(* IEC 61131-3 sources: eCockpitGit/test_project/src/%F%00 Library/%F%Common Functions/%F%Time, 12 files *)

(* ---- %DUT%ATimeShow.st ---- *)
TYPE ATimeShow : STRING(19); END_TYPE

(* ---- %POU%FU_sCountUpDateTime.st ---- *)
//This function, converts passed seconds to minutes, hours, days, weeks, years, and only outputs the two biggest active time formats
//example 249 = Minutes: 4 Seconds: 9, 529385 = Days: 6 Hours: 3
// |**Version**|**Author**| **Date** |**Changes**
// | 1         | NSN      | 09-01-18 | Updated to new format
// | 1         | NSN      | 13-06-18 | Updated names and types
FUNCTION FU_sCountUpDateTime : STRING(24)
VAR_INPUT
	dwSeconds	:DWORD;		//Input seconds
END_VAR
VAR
	Remains		:DWORD;		//Date time converted to seconds
	Buffer1		:DWORD;		//Buffer for first value
	Buffer2		:DWORD;		//Buffer for second value
END_VAR
(*%!%__DELIMITER__%!%*)
Remains 							:=		dwSeconds;
IF Remains < 604799 THEN
	IF Remains < 86401 THEN
		IF Remains < 3601 THEN
			IF Remains < 61 THEN	//This calculates the seconds
				Buffer1				:=		Remains;
				FU_sCountUpDateTime	:=		FU_sConcat('Seconds: ', TO_STRING(Buffer1));
			ELSE					//This calculates the minutes and seconds
				Buffer1				:=		Remains / 60;
				Remains				:=		(Remains - (Buffer1 * 60));
				Buffer2				:=		Remains;
				FU_sCountUpDateTime	:=		FU_sConcat('Minutes: ', TO_STRING(Buffer1));
				FU_sCountUpDateTime	:=		FU_sConcat(FU_sCountUpDateTime, ' Seconds: ');
				FU_sCountUpDateTime	:=		FU_sConcat(FU_sCountUpDateTime, TO_STRING(Buffer2));
			END_IF
		ELSE						//This calculates the hours and minutes
			Buffer1					:=		Remains / 3600;
			Remains					:=		(Remains - (Buffer1 * 3600));
			Buffer2					:=		Remains / 60;
			FU_sCountUpDateTime		:=		FU_sConcat('Hours: ', TO_STRING(Buffer1));
			FU_sCountUpDateTime		:=		FU_sConcat(FU_sCountUpDateTime, ' Minutes: ');
			FU_sCountUpDateTime		:=		FU_sConcat(FU_sCountUpDateTime, TO_STRING(Buffer2));
		END_IF
	ELSE							//This calculates the days and hours
		Buffer1						:=		Remains / 86400;
		Remains						:=		(Remains - (Buffer1 * 86400));
		Buffer2						:=		Remains / 3600;
		FU_sCountUpDateTime			:=		FU_sConcat('Days: ', TO_STRING(Buffer1));
		FU_sCountUpDateTime			:=		FU_sConcat(FU_sCountUpDateTime, ' Hours: ');
		FU_sCountUpDateTime			:=		FU_sConcat(FU_sCountUpDateTime, TO_STRING(Buffer2));
	END_IF
ELSE
	Buffer1							:=		Remains / 604800;
	Remains							:=		(Remains - (Buffer1 * 604800));
	Buffer2							:=		Remains / 86400;
	FU_sCountUpDateTime				:=		FU_sConcat('Weeks: ', TO_STRING(Buffer1));
	FU_sCountUpDateTime				:=		FU_sConcat(FU_sCountUpDateTime, ' Days: ');
	FU_sCountUpDateTime				:=		FU_sConcat(FU_sCountUpDateTime, TO_STRING(Buffer2));
END_IF

(* ---- %POU%FU_sDTToStringHH_MM_SS.st ---- *)
//This function extracts the time and date from a dt variable and outputs it as a string with the format hh:mm:ss
// |**Version**|**Author**| **Date** |**Changes**
// | 1         | NSN      | 14-06-18 | Creation
FUNCTION FU_sDTToStringHH_MM_SS: STRING(8)
VAR
	dtConv		:STRING(22);	//dt converted to a string
END_VAR
VAR_INPUT
	dtDateTime	:DT;			//The input dt
END_VAR
(*%!%__DELIMITER__%!%*)
dtConv									:=		TO_STRING(dtDateTime);		//The dt is converted to a string
FU_sDTToStringHH_MM_SS					:=		FU_sMID(dtConv,8,15);	//The string components are extracted

(* ---- %POU%FU_sDTToStringHH_MM_SS_DD_MM_YY.st ---- *)
//This function extracts the time and date from a dt variable and outputs it as a string with the format hh:mm:ss dd-mm-yy
// |**Version**|**Author**| **Date** |**Changes**
// | 1         | NSN      | 21-06-18 | Creation
FUNCTION FU_sDTToStringHH_MM_SS_DD_MM_YY: STRING(17)
VAR
	dtConv		:STRING(22);	//dt converted to a string
END_VAR
VAR_INPUT
	dtDateTime	:DT;			//The input dt
END_VAR
(*%!%__DELIMITER__%!%*)
dtConv									:=		TO_STRING(dtDateTime);		//The dt is converted to a string
FU_sDTToStringHH_MM_SS_DD_MM_YY			:=
FU_sConcat(
FU_sMID(dtConv,8,15)
,
FU_sConcat(' ',FU_sConcat(FU_sMID(dtConv,2,12),FU_sConcat(FU_sMID(dtConv,4,8),FU_sMID(dtConv,2,6))))
);	//The string components are extracted

(* ---- %POU%FU_sDTToStringHH_MM_SS_DD_MM_YYYY.st ---- *)
//This function extracts the time and date from a dt variable and outputs it as a string with the format hh:mm:ss dd-mm-yyyy
// |**Version**|**Author**| **Date** |**Changes**
// | 1         | NSN      | 21-06-18 | Creation
FUNCTION FU_sDTToStringHH_MM_SS_DD_MM_YYYY: STRING(19)
VAR
	dtConv		:STRING(22);	//dt converted to a string
END_VAR
VAR_INPUT
	dtDateTime	:DT;			//The input dt
END_VAR
(*%!%__DELIMITER__%!%*)
dtConv									:=		TO_STRING(dtDateTime);		//The dt is converted to a string
FU_sDTToStringHH_MM_SS_DD_MM_YYYY		:=
FU_sConcat(
FU_sMID(dtConv,8,15)
,
FU_sConcat(' ',FU_sConcat(FU_sMID(dtConv,2,12),FU_sConcat(FU_sMID(dtConv,4,8),FU_sMID(dtConv,4,4))))
);

(* ---- %POU%FU_sDTToStringHH_MM_SS_YY_MM_DD.st ---- *)
//This function extracts the time and date from a dt variable and outputs it as a string with the format hh:mm:ss yy-mm-dd
// |**Version**|**Author**| **Date** |**Changes**
// | 1         | NSN      | 05-04-18 | Creation
FUNCTION FU_sDTToStringHH_MM_SS_YY_MM_DD: STRING(17)
VAR
	dtConv		:STRING(22);	//dt converted to a string
END_VAR
VAR_INPUT
	dtDateTime	:DT;			//The input dt
END_VAR
(*%!%__DELIMITER__%!%*)
dtConv									:=		TO_STRING(dtDateTime);		//The dt is converted to a string
FU_sDTToStringHH_MM_SS_YY_MM_DD			:=		FU_sConcat(FU_sMID(dtConv,8,15),FU_sConcat(' ',FU_sMID(dtConv,8,6)));	//The string components are extracted

(* ---- %POU%FU_sDTToStringHH_MM_SS_YYYY_MM_DD.st ---- *)
//This function extracts the time and date from a dt variable and outputs it as a string with the format hh:mm:ss yyyy-mm-dd
// |**Version**|**Author**| **Date** |**Changes**
// | 1         | NSN      | 05-04-18 | Creation
FUNCTION FU_sDTToStringHH_MM_SS_YYYY_MM_DD: STRING(19)
VAR
	dtConv		:STRING(22);	//dt converted to a string
END_VAR
VAR_INPUT
	dtDateTime	:DT;			//The input dt
END_VAR
(*%!%__DELIMITER__%!%*)
dtConv									:=		TO_STRING(dtDateTime);		//The dt is converted to a string
FU_sDTToStringHH_MM_SS_YYYY_MM_DD		:=		FU_sConcat(FU_sMID(dtConv,8,15),FU_sConcat(' ',FU_sMID(dtConv,10,4)));	//The string components are extracted

(* ---- %POU%FU_sDTToStringSS_MM_HH_DD_MM_YY.st ---- *)
//This function extracts the time and date from a dt variable and outputs it as a string with the format hh:mm:ss yy-mm-dd
//DT#2018-04-26-15:56:48
// |**Version**|**Author**| **Date** |**Changes**
// | 1         | NSN      | 05-04-18 | Creation
FUNCTION FU_sDTToStringSS_MM_HH_DD_MM_YY: STRING(17)
VAR
	dtConv		:STRING(22);	//dt converted to a string
END_VAR
VAR_INPUT
	dtDateTime	:DT;			//The input dt
END_VAR
(*%!%__DELIMITER__%!%*)
dtConv									:=		TO_STRING(dtDateTime);		//The dt is converted to a string
FU_sDTToStringSS_MM_HH_DD_MM_YY			:=
FU_sConcat(

FU_sConcat(FU_sMID(dtConv,2,21),FU_sConcat(FU_sMID(dtConv,4,17),FU_sMID(dtConv,2,15)))

,

FU_sConcat(' ',FU_sConcat(FU_sMID(dtConv,2,12),FU_sConcat(FU_sMID(dtConv,4,8),FU_sMID(dtConv,2,6))))

);	//The string components are extracted

(* ---- %POU%FU_sDTToStringSS_MM_HH_DD_MM_YYYY.st ---- *)
//This function extracts the time and date from a dt variable and outputs it as a string with the format hh:mm:ss yyyy-mm-dd
// |**Version**|**Author**| **Date** |**Changes**
// | 1         | NSN      | 05-04-18 | Creation
FUNCTION FU_sDTToStringSS_MM_HH_DD_MM_YYYY: STRING(19)
VAR
	dtConv		:STRING(22);	//dt converted to a string
END_VAR
VAR_INPUT
	dtDateTime	:DT;			//The input dt
END_VAR
(*%!%__DELIMITER__%!%*)
dtConv									:=		TO_STRING(dtDateTime);		//The dt is converted to a string
FU_sDTToStringSS_MM_HH_DD_MM_YYYY		:=
FU_sConcat(
FU_sConcat(FU_sMID(dtConv,2,21),FU_sConcat(FU_sMID(dtConv,4,17),FU_sMID(dtConv,2,15)))

,

FU_sConcat(' ',FU_sConcat(FU_sMID(dtConv,2,12),FU_sConcat(FU_sMID(dtConv,4,8),FU_sMID(dtConv,4,4))))

);

(* ---- %POU%FU_sDTToStringYY_MM_DD_HH_MM_SS.st ---- *)
//This function extracts the time and date from a dt variable and outputs it as a string with the format yy-mm-dd hh:mm:ss
//DT#2018-4-26-15:56:48 --> 'DT#2018-04-26-16:04:54' --> '18-04-26 15:56:48'
// |**Version**|**Author**| **Date** |**Changes**
// | 1         | NSN      | 25-04-18 | Creation
FUNCTION FU_sDTToStringYY_MM_DD_HH_MM_SS: STRING(17)
VAR
	dtConv		:STRING(22);	//dt converted to a string
END_VAR
VAR_INPUT
	dtDateTime	:DT;			//The input dt
END_VAR
(*%!%__DELIMITER__%!%*)
dtConv							:=		TO_STRING(dtDateTime);		//The dt is converted to a string
FU_sDTToStringYY_MM_DD_HH_MM_SS	:=		FU_sConcat(FU_sMID(dtConv,8,6),FU_sConcat(' ',FU_sMID(dtConv,8,15)));			//The string components are extracted and combined

(* ---- %POU%FU_sDTToStringYYYY_MM_DD_HH_MM_SS.st ---- *)
//This function extracts the time and date from a dt variable and outputs it as a string with the format yyyy-mm-dd hh:mm:ss
//DT#2018-4-26-15:56:48 --> 'DT#2018-04-26-16:04:54' --> '2018-04-26-15:56:48'
// |**Version**|**Author**| **Date** |**Changes**
// | 1         | NSN      | 25-04-18 | Creation
// | 1         | NSN      | 16-09-20 | Changed 2018-04-26 15:56:48 to 2018-04-26-15:56:48 to reduce cpu usage
FUNCTION FU_sDTToStringYYYY_MM_DD_HH_MM_SS: STRING(19)
VAR
	dtConv		:STRING(22);	//dt converted to a string
END_VAR
VAR_INPUT
	dtDateTime	:DT;			//The input dt
END_VAR
(*%!%__DELIMITER__%!%*)
dtConv								:=		TO_STRING(dtDateTime);		//The dt is converted to a string
FU_sDTToStringYYYY_MM_DD_HH_MM_SS	:=		FU_sMidBI(sStr:=dtConv,wLen:=19,wPos:=4);			//The string components are extracted and combined

(* ---- %POU%FU_StringYYYY_MM_DD_HH_MM_SSToDT.st ---- *)
//This function converts a string with the format yyyy-mm-dd-hh:mm:ss to a dt
//DT#2018-4-26-15:56:48 --> 'DT#2018-04-26-16:04:54' --> '2018-04-26-15:56:48'
// |**Version**|**Author**| **Date** |**Changes**
// | 1         | NSN      | 16-09-20 | Creation
FUNCTION FU_StringYYYY_MM_DD_HH_MM_SSToDT: DT
VAR_INPUT
	str	:STRING(19);			//The input dt
END_VAR
(*%!%__DELIMITER__%!%*)
FU_StringYYYY_MM_DD_HH_MM_SSToDT	:=		TO_DT(FU_sConcat(s1:='DT#',s2:=str));			//The string components are extracted and combined
